// TIA Portal V20 export
TYPE "sAxis_Para"
   STRUCT
      rJog_Speed : Array[0..2] of LReal;   // 点动速度/ACC/DEC/JERK
      rMV_Speed : Array[0..2] of LReal;   // 速度运行速度/ACC/DEC/JERK
      rStop_Dec : Array[0..1] of LReal;
      rEStop_Dec : Array[0..1] of LReal;
      iNum_Abspos : Int := 4;
      rPos_Abs : Array[0..16] of LReal;   // 绝对定位目标位置 / Over travel switch set
      rSpeed_Abs : Array[0..16] of LReal;   // Endlage Unten / 绝对定位速度
      rAcc_Set : Array[0..16] of LReal;   // 绝对定位加速度 / Overtravel switch Reset
      rDec_Set : Array[0..16] of LReal;   // 绝对定位减速度 / Belt check sensor
      rJerk_Set : Array[0..16] of LReal;   // 绝对定位加加速度
      rSpeedPercent : LReal := 20.0;   // Endlage Unten / 速度设定百分比
      iHomeMode : Int;   // 回零方式
      rHomePos : LReal;   // 回零位置
   END_STRUCT;
   // rJog_Speed[0] := 10.0;
   // rJog_Speed[1..2] := 30.0;
   // rMV_Speed[0] := 20.0;
   // rMV_Speed[1..2] := 30.0;
   // rStop_Dec[0] := 30.0;
   // rStop_Dec[1] := 50.0;
   // rEStop_Dec[0..1] := 50.0;
   // rPos_Abs[1] := 10.0;
   // rPos_Abs[2] := 20.0;
   // rPos_Abs[3] := 30.0;
   // rPos_Abs[4] := 40.0;
   // rPos_Abs[5] := 50.0;
   // rPos_Abs[6] := 60.0;
   // rPos_Abs[7] := 70.0;
   // rPos_Abs[8] := 80.0;
   // rPos_Abs[9] := 90.0;
   // rPos_Abs[10] := 100.0;
   // rPos_Abs[11] := 110.0;
   // rPos_Abs[12] := 120.0;
   // rPos_Abs[13] := 130.0;
   // rPos_Abs[14] := 140.0;
   // rPos_Abs[15] := 150.0;
   // rPos_Abs[16] := 160.0;
   // rSpeed_Abs[0..16] := 20.0;
   // rAcc_Set[0..16] := 50.0;
   // rDec_Set[0..16] := 50.0;
   // rJerk_Set[0..16] := 50.0;
END_TYPE
